PROGRAM MAIN
VAR

	fbDestination :REFERENCE TO FB_DestinationDataStore;
	fbSource: REFERENCE TO DUT_SourceDataStore;
	nDestination: UINT;
	nSource: UINT;
	nIndex: UINT;
END_VAR

GVL_BTPS.fbBay1Linear(bEnable:=TRUE);
GVL_BTPS.fbBay3Linear(bEnable:=TRUE);
GVL_BTPS.fbBay4Linear(bEnable:=TRUE);

GVL_BTPS.fbBay1Rotary(bEnable:=TRUE);
GVL_BTPS.fbBay3Rotary(bEnable:=TRUE);
GVL_BTPS.fbBay4Rotary(bEnable:=TRUE);

GVL_BTPS.fbBay1Goniometer(bEnable:=TRUE);
GVL_BTPS.fbBay3Goniometer(bEnable:=TRUE);
GVL_BTPS.fbBay4Goniometer(bEnable:=TRUE);

GVL_BTPS.fbDestinations[1](sName:='TMO IP1', fbDestinationValve:=GVL_BTPS.fbDestinationValves[1]);
GVL_BTPS.fbDestinations[2](sName:='TMO IP2', fbDestinationValve:=GVL_BTPS.fbDestinationValves[2]);
GVL_BTPS.fbDestinations[3](sName:='TMO IP3', fbDestinationValve:=GVL_BTPS.fbDestinationValves[3]);
GVL_BTPS.fbDestinations[4](sName:='RIX qRIXS', fbDestinationValve:=GVL_BTPS.fbDestinationValves[4]);
GVL_BTPS.fbDestinations[5](sName:='RIX ChemRIXS', fbDestinationValve:=GVL_BTPS.fbDestinationValves[5]);
GVL_BTPS.fbDestinations[6](sName:='XPP', fbDestinationValve:=GVL_BTPS.fbDestinationValves[6]);
GVL_BTPS.fbDestinations[7](sName:='Laser Lab', fbDestinationValve:=GVL_BTPS.fbDestinationValves[7]);

END_PROGRAM

(* stored: Version 1.1.0.1, ProductVersion 3.1.4022.18
   POU MAIN: Id {98170510-de7b-424a-a18f-b4c889af69d0}, SpecialFunc None *)
